# EPICS substitutions: tests/test_parsers/examples/afg3011.substitutions
file TektronixAFG3K.template
{
pattern {P, R, PORT}
{"TST:", "AFG3011", "AFG3K"}
{"TST:", "AFG3011", "AFG3K2"}
}

file TektronixAFG3K_Output.template
{
pattern {P, R, PORT, OUTPUT_NUM}
{"TST:", "AFG3011:Output", "AFG3K", "1"}
}

file TektronixAFG3K_Source.template
{
pattern {P, R, PORT, SOURCE_NUM}
{"TST:", "AFG3011:Source", "AFG3K", "1"}
}
